Template "Vorlage_1" 800x420
   Button "Beenden" at 720,360 size 78x58; TextOff 'Beenden / Exit'; PictureOff "ExitRuntime_TP700_Comfort_TR"; PictureOn "ExitRuntime_TP700_Comfort_TR"
      on Release: StopRuntime(0)
   Button "Template_Button" at 640,360 size 78x58; TextOff 'Text'
   Button "Template_Button_1" at 560,360 size 78x58; TextOff 'Text'
   Button "Template_Button_2" at 480,360 size 78x58; TextOff 'Text'
   Button "Template_Button_3" at 400,360 size 78x58; TextOff 'Text'
   Button "Template_Button_4" at 321,360 size 78x58; TextOff 'Text'
   Button "Template_Button_5" at 241,360 size 78x58; TextOff 'Meldungen'
      on Click: function_ef3f5d25("Meldefenster_Anstehend", -1)
   Button "Template_Button_6" at 161,360 size 78x58; TextOff 'Übersicht'
      on Release: ActivateScreen("2_Übersicht", 0)
   Button "Template_Button_7" at 81,360 size 78x58; TextOff 'zurück'
      on Click: function_efd93a16()
   Button "Startbild" at 1,360 size 78x58; TextOff 'Startbild / Start screen'; PictureOff "NavigateHome_TP700_Comfort_TR"; PictureOn "NavigateHome_TP700_Comfort_TR"
      on Release: ActivateScreen("1_Grundbild", 0)
   AlarmView "Meldeanzeige_Nichtquittiert" at 0,0 size 800x20

screen "1_Grundbild" 800x420, template "Vorlage_1"
   on GenerateScreen: SetTag("Header_Line_1", 1)
   Button "HmiScreenItemData" at 36,60 size 159x47; TextOff 'Automatik'; PictureOff "Navigates to Automatik for TP700 Comfort 17.0.0.0"; PictureOn "Navigates to Automatik for TP700 Comfort 17.0.0.0"
      on Release: ActivateScreen("100_Automatik", 0)
   Button "HmiScreenItemData_1" at 36,119 size 159x47; TextOff 'Einrichten'; PictureOff "Navigates to Einrichten for TP700 Comfort 17.0.0.0"; PictureOn "Navigates to Einrichten for TP700 Comfort 17.0.0.0"
      on Release: ActivateScreen("10_Einrichten", 0)
   Button "HmiScreenItemData_3" at 36,178 size 159x47; TextOff 'Systembilder / System screens'; PictureOff "Navigates to Systembilder for TP700 Comfort 17.0.0.0"; PictureOn "Navigates to Systembilder for TP700 Comfort 17.0.0.0"
      on Release: ActivateScreen("1000_Systembilder", 0)

screen "100_Automatik" 800x420, template "Vorlage_1"
   on GenerateScreen: SetTag("Header_Line_1", 100)

screen "10_Einrichten" 800x420, template "Vorlage_1"
   on GenerateScreen: SetTag("Header_Line_1", 10)
   Button "HmiScreenItemData_1" at 35,41 size 159x47; TextOff 'FG 1 / Einrichtfunktionen'; TextOn 'Einrichtfunktionen'; PictureOff "Navigates to Einrichtfunktionen for TP700 Comfort 17.0.0.0"; PictureOn "Navigates to Einrichtfunktionen for TP700 Comfort 17.0.0.0"
      on Release: ActivateScreen("12_Einrichtfunktionen", 0); SetTag("HmiManualMovement_selection_station", 1)
      Visibility <- "exists"
   Button "HmiScreenItemData_2" at 35,100 size 159x47; TextOff 'FG 2 / Einrichtfunktionen'; TextOn 'Einrichtfunktionen'; PictureOff "Navigates to Einrichtfunktionen for TP700 Comfort 17.0.0.0"; PictureOn "Navigates to Einrichtfunktionen for TP700 Comfort 17.0.0.0"
      on Release: ActivateScreen("12_Einrichtfunktionen", 0); SetTag("HmiManualMovement_selection_station", 2)
      Visibility <- "exists"
   Button "HmiScreenItemData_3" at 35,160 size 159x47; TextOff 'FG 3 / Einrichtfunktionen'; TextOn 'Einrichtfunktionen'; PictureOff "Navigates to Einrichtfunktionen for TP700 Comfort 17.0.0.0"; PictureOn "Navigates to Einrichtfunktionen for TP700 Comfort 17.0.0.0"
      on Release: ActivateScreen("12_Einrichtfunktionen", 0); SetTag("HmiManualMovement_selection_station", 3)
      Visibility <- "exists"
   Button "HmiScreenItemData_4" at 35,223 size 159x47; TextOff 'FG 4 / Einrichtfunktionen'; TextOn 'Einrichtfunktionen'; PictureOff "Navigates to Einrichtfunktionen for TP700 Comfort 17.0.0.0"; PictureOn "Navigates to Einrichtfunktionen for TP700 Comfort 17.0.0.0"
      on Release: ActivateScreen("12_Einrichtfunktionen", 0); SetTag("HmiManualMovement_selection_station", 4)
      Visibility <- "exists"
   Button "HmiScreenItemData_5" at 35,282 size 159x47; TextOff 'FG 5 / Einrichtfunktionen'; TextOn 'Einrichtfunktionen'; PictureOff "Navigates to Einrichtfunktionen for TP700 Comfort 17.0.0.0"; PictureOn "Navigates to Einrichtfunktionen for TP700 Comfort 17.0.0.0"
      on Release: ActivateScreen("12_Einrichtfunktionen", 0); SetTag("HmiManualMovement_selection_station", 5)
      Visibility <- "exists"
   Button "HmiScreenItemData_6" at 232,282 size 159x47; TextOff 'FG Transport / Einrichtfunktionen'; TextOn 'Einrichtfunktionen'; PictureOff "Navigates to Einrichtfunktionen for TP700 Comfort 17.0.0.0"; PictureOn "Navigates to Einrichtfunktionen for TP700 Comfort 17.0.0.0"
      on Release: ActivateScreen("12_Einrichtfunktionen", 0); SetTag("HmiManualMovement_selection_station", 10)
      Visibility <- "exists"
   Button "HmiScreenItemData_7" at 232,41 size 159x47; TextOff 'FG 6 / Einrichtfunktionen'; TextOn 'Einrichtfunktionen'; PictureOff "Navigates to Einrichtfunktionen for TP700 Comfort 17.0.0.0"; PictureOn "Navigates to Einrichtfunktionen for TP700 Comfort 17.0.0.0"
      on Release: ActivateScreen("12_Einrichtfunktionen", 0); SetTag("HmiManualMovement_selection_station", 1)
      Visibility <- "exists"
   Button "HmiScreenItemData_8" at 232,100 size 159x47; TextOff 'FG 7 / Einrichtfunktionen'; TextOn 'Einrichtfunktionen'; PictureOff "Navigates to Einrichtfunktionen for TP700 Comfort 17.0.0.0"; PictureOn "Navigates to Einrichtfunktionen for TP700 Comfort 17.0.0.0"
      on Release: ActivateScreen("12_Einrichtfunktionen", 0); SetTag("HmiManualMovement_selection_station", 1)
      Visibility <- "exists"
   Button "HmiScreenItemData_9" at 232,159 size 159x47; TextOff 'FG 8 / Einrichtfunktionen'; TextOn 'Einrichtfunktionen'; PictureOff "Navigates to Einrichtfunktionen for TP700 Comfort 17.0.0.0"; PictureOn "Navigates to Einrichtfunktionen for TP700 Comfort 17.0.0.0"
      on Release: ActivateScreen("12_Einrichtfunktionen", 0); SetTag("HmiManualMovement_selection_station", 1)
      Visibility <- "exists"
   Button "HmiScreenItemData_10" at 232,218 size 159x47; TextOff 'FG 9 / Einrichtfunktionen'; TextOn 'Einrichtfunktionen'; PictureOff "Navigates to Einrichtfunktionen for TP700 Comfort 17.0.0.0"; PictureOn "Navigates to Einrichtfunktionen for TP700 Comfort 17.0.0.0"
      on Release: ActivateScreen("12_Einrichtfunktionen", 0); SetTag("HmiManualMovement_selection_station", 1)
      Visibility <- "exists"

screen "12_Einrichtfunktionen" 800x420, template "Vorlage_1"
   on GenerateScreen: SetTag("Header_Line_1", 12); SetTag("Header_Line_2", 1)
   on ClearScreen: SetTag("HmiManualMovement_selection_station", 0); SetTag("Header_Line_2", 0)
   Rectangle "recExecuteLeft1" at 0,22 size 285x72
      Visibility <- "showRecLeft"
   Rectangle "recRuntime1" at 287,22 size 226x72
      Visibility <- "showName"
   Rectangle "recExecuteRight1" at 515,22 size 285x72
      Visibility <- "showRecRight"
   Rectangle "recConfirmExecuteLeft1" at 60,26 size 29x29
      Appearance <- "workAct"
      Visibility <- "isExecutableLeft"
   Rectangle "recFinalPositionLeft1" at 60,61 size 29x29
      Appearance <- "inWorkPos"
      Visibility <- "hasEndPositionLeft"
   Polygon "polExecutabilityLeft1" at 2,30 size 51x55
      Appearance <- "workIsInterlocked"
      Visibility <- "isExecutableLeft"
   SymbolicIOField "seaConfirmExecuteLeft1" at 92,26 size 193x29; TextOn '1'; TextOff '0'; TextList "Setup"
      ProcessValue <- "textlistFunctionExecuteLeft"
      Visibility <- "isExecutableLeft"
   SymbolicIOField "seaFinalPositionLeft1" at 92,61 size 193x29; TextOn '1'; TextOff '0'; TextList "Setup"
      ProcessValue <- "textlistFunctionFinalPosLeft"
      Visibility <- "hasEndPositionLeft"
   Rectangle "recFinalPositionRight1" at 711,61 size 29x29
      Appearance <- "inHomePos"
      Visibility <- "hasEndPositionRight"
   Polygon "polExecutabilityRight1" at 747,30 size 51x55
      Appearance <- "homeIsInterlocked"
      Visibility <- "isExecutableRight"
   SymbolicIOField "seaFunction1" at 287,26 size 226x29; TextOn '1'; TextOff '0'; TextList "Setup"
      ProcessValue <- "textlistFunctionName"
      Visibility <- "showName"
   SymbolicIOField "seaConfirmExecuteRight1" at 515,26 size 193x29; TextOn '1'; TextOff '0'; TextList "Setup"
      ProcessValue <- "textlistFunctionExecuteRight"
      Visibility <- "isExecutableRight"
   SymbolicIOField "seaFinalPositionRight1" at 515,61 size 193x29; TextOn '1'; TextOff '0'; TextList "Setup"
      ProcessValue <- "textlistFunctionFinalPosRight"
      Visibility <- "hasEndPositionRight"
   IOField "eaPosition1" at 287,61 size 226x29; FormatPattern s999999999.999
      ProcessValue <- "value"
      Visibility <- "showValue"
   Rectangle "recConfirmExecuteRight1" at 711,26 size 29x29
      Appearance <- "homeAct"
      Visibility <- "isExecutableRight"
   Button "btnRight1" at 515,22 size 285x72; TextOn 'Texto / Texte / Testo / 文本 / Text / Szöv / Текст / Tekst'; TextOff 'Texto / Texte / Testo / 文本 / Text / Szöv / Текст / Tekst'
      on Release: SetTag("moveHomePos", 0)
      on Press: SetTag("moveHomePos", 1)
      ObjectEnable <- "isExecutableRight"
   Button "btnLeft1" at 0,22 size 285x72; TextOn 'Texto / Texte / Testo / 文本 / Text / Szöv / Текст / Tekst'; TextOff 'Texto / Texte / Testo / 文本 / Text / Szöv / Текст / Tekst'
      on Release: SetTag("moveWorkPos", 0)
      on Press: SetTag("moveWorkPos", 1)
      ObjectEnable <- "isExecutableLeft"
   TextField "txtPage" at 575,326 size 69x29; Text 'Seite / Página / Page / Pagina / 页 / Stránka / Oldal / Страница / stron / Sida / Pagină'
   IOField "eaActualPage" at 654,326 size 41x29; FormatPattern 999
      ProcessValue <- "HmiManualMovement_selection_page"
   TextField "txtOf" at 705,326 size 38x29; Text 'von / de / di / 之 / of / od / tól / из / z / av / din'
   IOField "eaNumberOfPages" at 753,326 size 41x29; FormatPattern 999
      ProcessValue <- "HmiManualMovement_selection_ofMaxPages"
   Group "Function 1" at 0,22 size 800x72; TextList "Setup"
   Group "Function 2" at 0,96 size 800x72; TextList "Setup"
   Group "Function 3" at 0,170 size 800x72; TextList "Setup"
   Group "Function 4" at 0,244 size 800x72; TextList "Setup"
   Button "Template_Button" at 640,360 size 78x58; TextOff 'Seite +'
      on Press: SetBit("HmiManualMovement_selection_nextPage")
   Button "Template_Button_1" at 560,360 size 78x58; TextOff 'Seite -'
      on Press: SetBit("HmiManualMovement_selection_previousPage")
   Button "Template_Button_2" at 480,360 size 78x58; TextOff 'Symbol Absolut'
      on Press: InvertBit("HmiManualMovement_selection_showSymbols")
   Rectangle "recExecuteLeft1_1" at 0,96 size 285x72
      Visibility <- "showRecLeft"
   Rectangle "recRuntime1_1" at 287,96 size 226x72
      Visibility <- "showName"
   Rectangle "recExecuteRight1_1" at 515,96 size 285x72
      Visibility <- "showRecRight"
   Rectangle "recConfirmExecuteLeft1_1" at 60,100 size 29x29
      Appearance <- "workAct"
      Visibility <- "isExecutableLeft"
   Rectangle "recFinalPositionLeft1_1" at 60,135 size 29x29
      Appearance <- "inWorkPos"
      Visibility <- "hasEndPositionLeft"
   Polygon "polExecutabilityLeft1_1" at 2,104 size 51x55
      Appearance <- "workIsInterlocked"
      Visibility <- "isExecutableLeft"
   SymbolicIOField "seaConfirmExecuteLeft1_1" at 92,100 size 193x29; TextOn '1'; TextOff '0'; TextList "Setup"
      ProcessValue <- "textlistFunctionExecuteLeft"
      Visibility <- "isExecutableLeft"
   SymbolicIOField "seaFinalPositionLeft1_1" at 92,135 size 193x29; TextOn '1'; TextOff '0'; TextList "Setup"
      ProcessValue <- "textlistFunctionFinalPosLeft"
      Visibility <- "hasEndPositionLeft"
   Rectangle "recFinalPositionRight1_1" at 711,135 size 29x29
      Appearance <- "inHomePos"
      Visibility <- "hasEndPositionRight"
   Polygon "polExecutabilityRight1_1" at 747,104 size 51x55
      Appearance <- "homeIsInterlocked"
      Visibility <- "isExecutableRight"
   SymbolicIOField "seaFunction1_1" at 287,100 size 226x29; TextOn '1'; TextOff '0'; TextList "Setup"
      ProcessValue <- "textlistFunctionName"
      Visibility <- "showName"
   SymbolicIOField "seaConfirmExecuteRight1_1" at 515,100 size 193x29; TextOn '1'; TextOff '0'; TextList "Setup"
      ProcessValue <- "textlistFunctionExecuteRight"
      Visibility <- "isExecutableRight"
   SymbolicIOField "seaFinalPositionRight1_1" at 515,135 size 193x29; TextOn '1'; TextOff '0'; TextList "Setup"
      ProcessValue <- "textlistFunctionFinalPosRight"
      Visibility <- "hasEndPositionRight"
   IOField "eaPosition1_1" at 287,135 size 226x29; FormatPattern s999999999.999
      ProcessValue <- "value"
      Visibility <- "showValue"
   Rectangle "recConfirmExecuteRight1_1" at 711,100 size 29x29
      Appearance <- "homeAct"
      Visibility <- "isExecutableRight"
   Button "btnRight1_1" at 515,96 size 285x72; TextOn 'Texto / Texte / Testo / 文本 / Text / Szöv / Текст / Tekst'; TextOff 'Texto / Texte / Testo / 文本 / Text / Szöv / Текст / Tekst'
      on Release: SetTag("moveHomePos", 0)
      on Press: SetTag("moveHomePos", 1)
      ObjectEnable <- "isExecutableRight"
   Button "btnLeft1_1" at 0,96 size 285x72; TextOn 'Texto / Texte / Testo / 文本 / Text / Szöv / Текст / Tekst'; TextOff 'Texto / Texte / Testo / 文本 / Text / Szöv / Текст / Tekst'
      on Release: SetTag("moveWorkPos", 0)
      on Press: SetTag("moveWorkPos", 1)
      ObjectEnable <- "isExecutableLeft"
   Rectangle "recExecuteLeft1_2" at 0,170 size 285x72
      Visibility <- "showRecLeft"
   Rectangle "recRuntime1_2" at 287,170 size 226x72
      Visibility <- "showName"
   Rectangle "recExecuteRight1_2" at 515,170 size 285x72
      Visibility <- "showRecRight"
   Rectangle "recConfirmExecuteLeft1_2" at 60,174 size 29x29
      Appearance <- "workAct"
      Visibility <- "isExecutableLeft"
   Rectangle "recFinalPositionLeft1_2" at 60,209 size 29x29
      Appearance <- "inWorkPos"
      Visibility <- "hasEndPositionLeft"
   Polygon "polExecutabilityLeft1_2" at 2,178 size 51x55
      Appearance <- "workIsInterlocked"
      Visibility <- "isExecutableLeft"
   SymbolicIOField "seaConfirmExecuteLeft1_2" at 92,174 size 193x29; TextOn '1'; TextOff '0'; TextList "Setup"
      ProcessValue <- "textlistFunctionExecuteLeft"
      Visibility <- "isExecutableLeft"
   SymbolicIOField "seaFinalPositionLeft1_2" at 92,209 size 193x29; TextOn '1'; TextOff '0'; TextList "Setup"
      ProcessValue <- "textlistFunctionFinalPosLeft"
      Visibility <- "hasEndPositionLeft"
   Rectangle "recFinalPositionRight1_2" at 711,209 size 29x29
      Appearance <- "inHomePos"
      Visibility <- "hasEndPositionRight"
   Polygon "polExecutabilityRight1_2" at 747,178 size 51x55
      Appearance <- "homeIsInterlocked"
      Visibility <- "isExecutableRight"
   SymbolicIOField "seaFunction1_2" at 287,174 size 226x29; TextOn '1'; TextOff '0'; TextList "Setup"
      ProcessValue <- "textlistFunctionName"
      Visibility <- "showName"
   SymbolicIOField "seaConfirmExecuteRight1_2" at 515,174 size 193x29; TextOn '1'; TextOff '0'; TextList "Setup"
      ProcessValue <- "textlistFunctionExecuteRight"
      Visibility <- "isExecutableRight"
   SymbolicIOField "seaFinalPositionRight1_2" at 515,209 size 193x29; TextOn '1'; TextOff '0'; TextList "Setup"
      ProcessValue <- "textlistFunctionFinalPosRight"
      Visibility <- "hasEndPositionRight"
   IOField "eaPosition1_2" at 287,209 size 226x29; FormatPattern s999999999.999
      ProcessValue <- "value"
      Visibility <- "showValue"
   Rectangle "recConfirmExecuteRight1_2" at 711,174 size 29x29
      Appearance <- "homeAct"
      Visibility <- "isExecutableRight"
   Button "btnRight1_2" at 515,170 size 285x72; TextOn 'Texto / Texte / Testo / 文本 / Text / Szöv / Текст / Tekst'; TextOff 'Texto / Texte / Testo / 文本 / Text / Szöv / Текст / Tekst'
      on Release: SetTag("moveHomePos", 0)
      on Press: SetTag("moveHomePos", 1)
      ObjectEnable <- "isExecutableRight"
   Button "btnLeft1_2" at 0,170 size 285x72; TextOn 'Texto / Texte / Testo / 文本 / Text / Szöv / Текст / Tekst'; TextOff 'Texto / Texte / Testo / 文本 / Text / Szöv / Текст / Tekst'
      on Release: SetTag("moveWorkPos", 0)
      on Press: SetTag("moveWorkPos", 1)
      ObjectEnable <- "isExecutableLeft"
   Rectangle "recExecuteLeft1_3" at 0,244 size 285x72
      Visibility <- "showRecLeft"
   Rectangle "recRuntime1_3" at 287,244 size 226x72
      Visibility <- "showName"
   Rectangle "recExecuteRight1_3" at 515,244 size 285x72
      Visibility <- "showRecRight"
   Rectangle "recConfirmExecuteLeft1_3" at 60,248 size 29x29
      Appearance <- "workAct"
      Visibility <- "isExecutableLeft"
   Rectangle "recFinalPositionLeft1_3" at 60,283 size 29x29
      Appearance <- "inWorkPos"
      Visibility <- "hasEndPositionLeft"
   Polygon "polExecutabilityLeft1_3" at 2,252 size 51x55
      Appearance <- "workIsInterlocked"
      Visibility <- "isExecutableLeft"
   SymbolicIOField "seaConfirmExecuteLeft1_3" at 92,248 size 193x29; TextOn '1'; TextOff '0'; TextList "Setup"
      ProcessValue <- "textlistFunctionExecuteLeft"
      Visibility <- "isExecutableLeft"
   SymbolicIOField "seaFinalPositionLeft1_3" at 92,283 size 193x29; TextOn '1'; TextOff '0'; TextList "Setup"
      ProcessValue <- "textlistFunctionFinalPosLeft"
      Visibility <- "hasEndPositionLeft"
   Rectangle "recFinalPositionRight1_3" at 711,283 size 29x29
      Appearance <- "inHomePos"
      Visibility <- "hasEndPositionRight"
   Polygon "polExecutabilityRight1_3" at 747,252 size 51x55
      Appearance <- "homeIsInterlocked"
      Visibility <- "isExecutableRight"
   SymbolicIOField "seaFunction1_3" at 287,248 size 226x29; TextOn '1'; TextOff '0'; TextList "Setup"
      ProcessValue <- "textlistFunctionName"
      Visibility <- "showName"
   SymbolicIOField "seaConfirmExecuteRight1_3" at 515,248 size 193x29; TextOn '1'; TextOff '0'; TextList "Setup"
      ProcessValue <- "textlistFunctionExecuteRight"
      Visibility <- "isExecutableRight"
   SymbolicIOField "seaFinalPositionRight1_3" at 515,283 size 193x29; TextOn '1'; TextOff '0'; TextList "Setup"
      ProcessValue <- "textlistFunctionFinalPosRight"
      Visibility <- "hasEndPositionRight"
   IOField "eaPosition1_3" at 287,283 size 226x29; FormatPattern s999999999.999
      ProcessValue <- "value"
      Visibility <- "showValue"
   Rectangle "recConfirmExecuteRight1_3" at 711,248 size 29x29
      Appearance <- "homeAct"
      Visibility <- "isExecutableRight"
   Button "btnRight1_3" at 515,244 size 285x72; TextOn 'Texto / Texte / Testo / 文本 / Text / Szöv / Текст / Tekst'; TextOff 'Texto / Texte / Testo / 文本 / Text / Szöv / Текст / Tekst'
      on Release: SetTag("moveHomePos", 0)
      on Press: SetTag("moveHomePos", 1)
      ObjectEnable <- "isExecutableRight"
   Button "btnLeft1_3" at 0,244 size 285x72; TextOn 'Texto / Texte / Testo / 文本 / Text / Szöv / Текст / Tekst'; TextOff 'Texto / Texte / Testo / 文本 / Text / Szöv / Текст / Tekst'
      on Release: SetTag("moveWorkPos", 0)
      on Press: SetTag("moveWorkPos", 1)
      ObjectEnable <- "isExecutableLeft"

screen "1000_Systembilder" 800x420, template "Vorlage_1"
   on GenerateScreen: SetTag("Header_Line_1", 1000)
   Button "Zurück" at 1,25 size 159x47; TextOff 'Zurück / Back'
      on Release: ActivateScreen("1_Grundbild", 0)
   Button "HmiScreenItemData" at 36,119 size 159x47; TextOff 'SIMATIC PLC Systemdiagnose SIMATIC PLC system diagnos...'; PictureOff "Navigates to SIMATIC PLC Systemdiagnose for TP700 Comfort 17.0.0.0"; PictureOn "Navigates to SIMATIC PLC Systemdiagnose for TP700 Comfort 17.0.0.0"
      on Release: ActivateScreen("1001_SIMATIC PLC Systemdiagnose", 0)
   Button "HmiScreenItemData_1" at 36,178 size 159x47; TextOff 'Projektinformatio nen Project information'; PictureOff "Navigates to Projektinformationen for TP700 Comfort 17.0.0.0"; PictureOn "Navigates to Projektinformationen for TP700 Comfort 17.0.0.0"
      on Release: ActivateScreen("1002_Projektinformationen", 0)
   Button "HmiScreenItemData_2" at 36,237 size 159x47; TextOff 'Systemeinstellung en System settings'; PictureOff "Navigates to Systemeinstellungen for TP700 Comfort 17.0.0.0"; PictureOn "Navigates to Systemeinstellungen for TP700 Comfort 17.0.0.0"
      on Release: ActivateScreen("1003_Systemeinstellungen", 0)
   Button "HmiScreenItemData_3" at 36,296 size 159x47; TextOff 'Benutzerverwaltu ng User administration'; PictureOff "Navigates to Benutzerverwaltung for TP700 Comfort 17.0.0.0"; PictureOn "Navigates to Benutzerverwaltung for TP700 Comfort 17.0.0.0"
      on Release: ActivateScreen("1004_Benutzerverwaltung", 0)
   Button "HmiScreenItemData_4" at 207,119 size 159x47; TextOff 'Systeminformatio nen System information'; PictureOff "Navigates to Systeminformationen for TP700 Comfort 17.0.0.0"; PictureOn "Navigates to Systeminformationen for TP700 Comfort 17.0.0.0"
      on Release: ActivateScreen("1005_Systeminformationen", 0)
   Button "HmiScreenItemData_5" at 207,178 size 159x47; TextOff 'Verschiedene Aufgaben Different jobs'; PictureOff "Navigates to Verschiedene Aufgaben for TP700 Comfort 17.0.0.0"; PictureOn "Navigates to Verschiedene Aufgaben for TP700 Comfort 17.0.0.0"
      on Release: ActivateScreen("1006_Verschiedene Aufgaben", 0)

screen "1001_SIMATIC PLC Systemdiagnose" 800x420, template "Vorlage_1"
   on GenerateScreen: SetTag("Header_Line_1", 1001)
   SysDiagControl "HmiScreenItemData" at 1,73 size 796x280
   Button "Zurück" at 1,25 size 159x47; TextOff 'Zurück / Back'
      on Release: ActivateScreen("1000_Systembilder", 0)

screen "1002_Projektinformationen" 800x420, template "Vorlage_1"
   on GenerateScreen: SetTag("Header_Line_1", 1002)
   TextField "HmiScreenItemData" at 35,75 size 171x28; Text 'Projektname: / Project name:'
   TextField "HmiScreenItemData_1" at 241,75 size 524x28; Text 'Demo-Projekt / Testprojekt_RV'
   TextField "HmiScreenItemData_2" at 35,105 size 171x28; Text 'Erstellt: / Created on:'
   TextField "HmiScreenItemData_3" at 241,105 size 524x28; Text '09.09.2024 14:49:17'
   TextField "HmiScreenItemData_4" at 35,135 size 171x28; Text 'Autor: / Author:'
   TextField "HmiScreenItemData_5" at 241,135 size 524x28; Text 'Andreas Fast Automation / AFA'
   TextField "HmiScreenItemData_6" at 35,165 size 171x28; Text 'Beschreibung: / Description:'
   TextField "HmiScreenItemData_7" at 241,165 size 524x28; Text '(nicht konfiguriert) / (not configured)'
   Button "Zurück" at 1,25 size 159x47; TextOff 'Zurück / Back'
      on Release: ActivateScreen("1000_Systembilder", 0)

screen "1003_Systemeinstellungen" 800x420, template "Vorlage_1"
   on GenerateScreen: SetTag("Header_Line_1", 1003)
   Button "Bildschirm kalibrieren" at 36,119 size 159x47; TextOff 'Bildschirm kalibri... / Calibrate screen'
      on Release: function_bc3e350c()
   Button "Putzbild" at 36,178 size 159x47; TextOff 'Putzbild / Clean screen'
      on Release: function_be740847(30)
   Button "Zurück" at 1,25 size 159x47; TextOff 'Zurück / Back'
      on Release: ActivateScreen("1000_Systembilder", 0)

screen "1004_Benutzerverwaltung" 800x420, template "Vorlage_1"
   on GenerateScreen: SetTag("Header_Line_1", 1004)
   UserView "HmiScreenItemData" at 1,73 size 796x280
   Button "Zurück" at 1,25 size 159x47; TextOff 'Zurück / Back'
      on Release: ActivateScreen("1000_Systembilder", 0)

screen "1005_Systeminformationen" 800x420, template "Vorlage_1"
   on GenerateScreen: SetTag("Header_Line_1", 1005)
   TextField "HmiScreenItemData" at 35,75 size 171x28; Text 'Bediengerätetyp: / HMI device type:'
   TextField "HmiScreenItemData_1" at 241,75 size 524x28; Text 'TP700 Comfort 17.0.0.0'
   TextField "HmiScreenItemData_2" at 35,105 size 171x28; Text 'Version:'
   TextField "HmiScreenItemData_3" at 35,135 size 171x28; Text 'Verbindung: / Connection:'
   TextField "HmiScreenItemData_4" at 241,135 size 524x28; Text 'ETHERNET'
   TextField "HmiScreenItemData_5" at 35,165 size 171x28; Text 'Steuerung: / PLC:'
   TextField "HmiScreenItemData_6" at 241,165 size 524x28; Text 'SIMATIC S7 1500'
   Button "Version anzeigen" at 241,105 size 524x28; TextOff 'Version anzeigen / Display version'
      on Release: function_febcb963(-1)
   Button "Zurück" at 1,25 size 159x47; TextOff 'Zurück / Back'
      on Release: ActivateScreen("1000_Systembilder", 0)

screen "1006_Verschiedene Aufgaben" 800x420, template "Vorlage_1"
   on GenerateScreen: SetTag("Header_Line_1", 1006)
   Button "Online" at 36,119 size 159x47; TextOff 'Online'
      on Release: function_bb44b551(0)
   Button "Offline" at 36,178 size 159x47; TextOff 'Offline'
      on Release: function_bb44b551(1)
   Button "Transfer" at 36,237 size 159x47; TextOff 'Transfer'
      on Release: function_bb44b551(2)
   Button "Sprache umschalten" at 36,296 size 159x47; TextOff 'Sprache umschal... / Toggle language'
      on Release: function_fb9197e8(-1)
   Button "Systemsteuerung" at 207,119 size 159x47; TextOff 'Systemsteuerung / Control Panel'
      on Release: function_f34a74f3()
   Button "Runtime beenden" at 207,178 size 159x47; TextOff 'Runtime beenden / Stop Runtime'
      on Release: StopRuntime(0)
   Button "Zurück" at 1,25 size 159x47; TextOff 'Zurück / Back'
      on Release: ActivateScreen("1000_Systembilder", 0)

screen "2_Übersicht" 800x420, template "Vorlage_1"
   on GenerateScreen: SetTag("Header_Line_1", 2)
   SymbolicIOField "Symbolisches_EA_Feld_Bild" at 47,80 size 365x42; TextOff '0'; TextOn '1'; TextList "Overview"
      ProcessValue <- "Übersicht_Station1"
   GraphicIOField "Vorlage_Grafisches EA-Feld_3" at 499,79 size 42x42; PictureOff "manual_off"; PictureOn "manual_on"
      ProcessValue <- "modeSetup"
   GraphicIOField "Vorlage_Grafisches EA-Feld_5" at 585,79 size 42x42; PictureOff "home_off"; PictureOn "home_on"
      ProcessValue <- "isInHome"
   GraphicIOField "Vorlage_Grafisches EA-Feld_6" at 628,79 size 42x42; PictureOff "homing_off"; PictureOn "homing_on"
      ProcessValue <- "isHoming"
   GraphicIOField "Vorlage_Grafisches EA-Feld_7" at 671,79 size 42x42; PictureOff "autoIsStopping_off"; PictureOn "autoIsStopping_on_blue"
      ProcessValue <- "autoIsStoping"
   SymbolicIOField "Symbolisches_EA_Feld_Bild_1" at 47,124 size 365x42; TextOff '0'; TextOn '1'; TextList "Overview"
      ProcessValue <- "Übersicht_Station2"
   GraphicIOField "Vorlage_Grafisches EA-Feld_8" at 413,123 size 42x42; PictureOff "auto_off"; PictureOn "auto_on"
      ProcessValue <- "modeAuto"
   GraphicIOField "Vorlage_Grafisches EA-Feld_9" at 456,123 size 42x42; PictureOff "step_off"; PictureOn "step_on"
      ProcessValue <- "modeTap"
   GraphicIOField "Vorlage_Grafisches EA-Feld_10" at 499,123 size 42x42; PictureOff "manual_off"; PictureOn "manual_on"
      ProcessValue <- "modeSetup"
   GraphicIOField "Vorlage_Grafisches EA-Feld_11" at 542,123 size 42x42; PictureOff "cycle_off"; PictureOn "cycle_on"
      ProcessValue <- "releaseCycle"
   GraphicIOField "Vorlage_Grafisches EA-Feld_12" at 585,123 size 42x42; PictureOff "home_off"; PictureOn "home_on"
      ProcessValue <- "isInHome"
   GraphicIOField "Vorlage_Grafisches EA-Feld_13" at 628,123 size 42x42; PictureOff "homing_off"; PictureOn "homing_on"
      ProcessValue <- "isHoming"
   GraphicIOField "Vorlage_Grafisches EA-Feld_14" at 671,123 size 42x42; PictureOff "autoIsStopping_off"; PictureOn "autoIsStopping_on_blue"
      ProcessValue <- "autoIsStoping"
   SymbolicIOField "Symbolisches_EA_Feld_Bild_2" at 47,168 size 365x42; TextOff '0'; TextOn '1'; TextList "Overview"
      ProcessValue <- "Übersicht_Station3"
   GraphicIOField "Vorlage_Grafisches EA-Feld_15" at 413,167 size 42x42; PictureOff "auto_off"; PictureOn "auto_on"
      ProcessValue <- "modeAuto"
   GraphicIOField "Vorlage_Grafisches EA-Feld_16" at 456,167 size 42x42; PictureOff "step_off"; PictureOn "step_on"
      ProcessValue <- "modeTap"
   GraphicIOField "Vorlage_Grafisches EA-Feld_17" at 499,167 size 42x42; PictureOff "manual_off"; PictureOn "manual_on"
      ProcessValue <- "modeSetup"
   GraphicIOField "Vorlage_Grafisches EA-Feld_18" at 542,167 size 42x42; PictureOff "cycle_off"; PictureOn "cycle_on"
      ProcessValue <- "releaseCycle"
   GraphicIOField "Vorlage_Grafisches EA-Feld_19" at 585,167 size 42x42; PictureOff "home_off"; PictureOn "home_on"
      ProcessValue <- "isInHome"
   GraphicIOField "Vorlage_Grafisches EA-Feld_20" at 628,167 size 42x42; PictureOff "homing_off"; PictureOn "homing_on"
      ProcessValue <- "isHoming"
   GraphicIOField "Vorlage_Grafisches EA-Feld_21" at 671,167 size 42x42; PictureOff "autoIsStopping_off"; PictureOn "autoIsStopping_on_blue"
      ProcessValue <- "autoIsStoping"
   SymbolicIOField "Symbolisches_EA_Feld_Bild_3" at 47,212 size 365x42; TextOff '0'; TextOn '1'; TextList "Overview"
      ProcessValue <- "Übersicht_Station4"
   GraphicIOField "Vorlage_Grafisches EA-Feld_22" at 413,211 size 42x42; PictureOff "auto_off"; PictureOn "auto_on"
      ProcessValue <- "modeAuto"
   GraphicIOField "Vorlage_Grafisches EA-Feld_23" at 456,211 size 42x42; PictureOff "step_off"; PictureOn "step_on"
      ProcessValue <- "modeTap"
   GraphicIOField "Vorlage_Grafisches EA-Feld_24" at 499,211 size 42x42; PictureOff "manual_off"; PictureOn "manual_on"
      ProcessValue <- "modeSetup"
   GraphicIOField "Vorlage_Grafisches EA-Feld_25" at 542,211 size 42x42; PictureOff "cycle_off"; PictureOn "cycle_on"
      ProcessValue <- "releaseCycle"
   GraphicIOField "Vorlage_Grafisches EA-Feld_26" at 585,211 size 42x42; PictureOff "home_off"; PictureOn "home_on"
      ProcessValue <- "isInHome"
   GraphicIOField "Vorlage_Grafisches EA-Feld_27" at 628,211 size 42x42; PictureOff "homing_off"; PictureOn "homing_on"
      ProcessValue <- "isHoming"
   GraphicIOField "Vorlage_Grafisches EA-Feld_28" at 671,211 size 42x42; PictureOff "autoIsStopping_off"; PictureOn "autoIsStopping_on_blue"
      ProcessValue <- "autoIsStoping"
   SymbolicIOField "Symbolisches_EA_Feld_Bild_4" at 47,256 size 365x42; TextOff '0'; TextOn '1'; TextList "Overview"
      ProcessValue <- "Übersicht_Station5"
   GraphicIOField "Vorlage_Grafisches EA-Feld_29" at 413,255 size 42x42; PictureOff "auto_off"; PictureOn "auto_on"
      ProcessValue <- "modeAuto"
   GraphicIOField "Vorlage_Grafisches EA-Feld_30" at 456,255 size 42x42; PictureOff "step_off"; PictureOn "step_on"
      ProcessValue <- "modeTap"
   GraphicIOField "Vorlage_Grafisches EA-Feld_31" at 499,255 size 42x42; PictureOff "manual_off"; PictureOn "manual_on"
      ProcessValue <- "modeSetup"
   GraphicIOField "Vorlage_Grafisches EA-Feld_32" at 542,255 size 42x42; PictureOff "cycle_off"; PictureOn "cycle_on"
      ProcessValue <- "releaseCycle"
   GraphicIOField "Vorlage_Grafisches EA-Feld_33" at 585,255 size 42x42; PictureOff "home_off"; PictureOn "home_on"
      ProcessValue <- "isInHome"
   GraphicIOField "Vorlage_Grafisches EA-Feld_34" at 628,255 size 42x42; PictureOff "homing_off"; PictureOn "homing_on"
      ProcessValue <- "isHoming"
   GraphicIOField "Vorlage_Grafisches EA-Feld_35" at 671,255 size 42x42; PictureOff "autoIsStopping_off"; PictureOn "autoIsStopping_on_blue"
      ProcessValue <- "autoIsStoping"
   SymbolicIOField "Symbolisches_EA_Feld_Bild_5" at 47,300 size 365x42; TextOff '0'; TextOn '1'; TextList "Overview"
      ProcessValue <- "Übersicht_Station10"
   GraphicIOField "Vorlage_Grafisches EA-Feld_36" at 413,299 size 42x42; PictureOff "auto_off"; PictureOn "auto_on"
      ProcessValue <- "modeAuto"
   GraphicIOField "Vorlage_Grafisches EA-Feld_37" at 456,299 size 42x42; PictureOff "step_off"; PictureOn "step_on"
      ProcessValue <- "modeTap"
   GraphicIOField "Vorlage_Grafisches EA-Feld_38" at 499,299 size 42x42; PictureOff "manual_off"; PictureOn "manual_on"
      ProcessValue <- "modeSetup"
   GraphicIOField "Vorlage_Grafisches EA-Feld_39" at 542,299 size 42x42; PictureOff "cycle_off"; PictureOn "cycle_on"
      ProcessValue <- "releaseCycle"
   GraphicIOField "Vorlage_Grafisches EA-Feld_40" at 585,299 size 42x42; PictureOff "home_off"; PictureOn "home_on"
      ProcessValue <- "isInHome"
   GraphicIOField "Vorlage_Grafisches EA-Feld_41" at 628,299 size 42x42; PictureOff "homing_off"; PictureOn "homing_on"
      ProcessValue <- "isHoming"
   GraphicIOField "Vorlage_Grafisches EA-Feld_42" at 671,299 size 42x42; PictureOff "autoIsStopping_off"; PictureOn "autoIsStopping_on_blue"
      ProcessValue <- "autoIsStoping"
   Switch "Schalter_1" at 414,80 size 42x42; CaptionText 'Switch'; TextOff 'OFF'; TextOn 'ON'; PictureOff "auto_off"; PictureOn "auto_on"
      ProcessValue <- "modeAuto"
   Switch "Schalter_2" at 457,80 size 42x42; CaptionText 'Switch'; TextOff 'OFF'; TextOn 'ON'; PictureOff "step_off"; PictureOn "step_on"
      ProcessValue <- "modeTap"
   Switch "Schalter_3" at 543,80 size 42x42; CaptionText 'Switch'; TextOff 'OFF'; TextOn 'ON'; PictureOff "cycle_off"; PictureOn "cycle_on"
      ProcessValue <- "releaseCycle"
   GraphicIOField "Vorlage_Grafisches EA-Feld_1" at 714,79 size 42x42; PictureOff "fault_off"; PictureOn "fault_on"
      ProcessValue <- "isInError"
   GraphicIOField "Vorlage_Grafisches EA-Feld_2" at 714,123 size 42x42; PictureOff "fault_off"; PictureOn "fault_on"
      ProcessValue <- "isInError"
   GraphicIOField "Vorlage_Grafisches EA-Feld_4" at 714,167 size 42x42; PictureOff "fault_off"; PictureOn "fault_on"
      ProcessValue <- "isInError"
   GraphicIOField "Vorlage_Grafisches EA-Feld_43" at 714,211 size 42x42; PictureOff "fault_off"; PictureOn "fault_on"
      ProcessValue <- "isInError"
   GraphicIOField "Vorlage_Grafisches EA-Feld_44" at 714,255 size 42x42; PictureOff "fault_off"; PictureOn "fault_on"
      ProcessValue <- "isInError"
   GraphicIOField "Vorlage_Grafisches EA-Feld_45" at 714,299 size 42x42; PictureOff "fault_off"; PictureOn "fault_on"
      ProcessValue <- "isInError"
   TextField "Textfeld_1" at 47,28 size 365x42; Text 'Maschine'
   GraphicIOField "Vorlage_Grafisches EA-Feld_46" at 413,28 size 42x42; PictureOff "manual_on"; PictureOn "auto_on"
      ProcessValue <- "automaticMode"
   Switch "Schalter_4" at 543,28 size 42x42; CaptionText 'Switch'; TextOff 'OFF'; TextOn 'ON'; PictureOff "cycle_off"; PictureOn "cycle_on"
      ProcessValue <- "automaticIsRunning"
   GraphicIOField "Vorlage_Grafisches EA-Feld_47" at 585,27 size 42x42; PictureOff "home_off"; PictureOn "home_on"
      ProcessValue <- "isInHome"
   GraphicIOField "Vorlage_Grafisches EA-Feld_48" at 628,27 size 42x42; PictureOff "homing_off"; PictureOn "homing_on"
      ProcessValue <- "isHoming"
   GraphicIOField "Vorlage_Grafisches EA-Feld_49" at 671,27 size 42x42; PictureOff "autoIsStopping_off"; PictureOn "autoIsStopping_on_blue"
      ProcessValue <- "automaticStops"
   GraphicIOField "Vorlage_Grafisches EA-Feld_50" at 714,27 size 42x42; PictureOff "fault_off"; PictureOn "fault_on"
      ProcessValue <- "isInError"
*)